{attribute 'qualified_only'}
TYPE PANotifyState :
(
	Off := 0,
	InfoOrActive := 1,
	AlarmOrFault := 2
);
END_TYPE

(* stored: Version 1.1.0.1, ProductVersion 3.1.4020.12
   DUT PANotifyState: Id {a7829e10-9170-42d6-9eb5-ee39942cfca0} *)
